PROGRAM ldrMain
VAR


	AIN1 AT %I*: UINT :=0;
	AOUT1 AT %Q*: INT := 1000;
	
	RUNNING: BOOL := FALSE;
	START: BOOL := TRUE;
	
END_VAR
VAR // added by the converter: edge detectors and wires of the graphical bodies
    _w1 : BOOL;
END_VAR

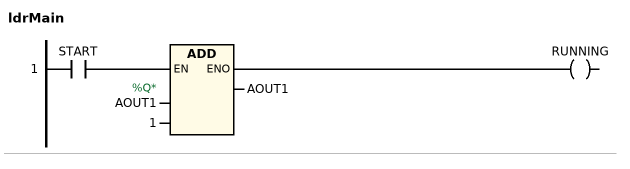
// NETWORK 1
//   AOUT1: AT %Q*
_w1 := START;
IF _w1 THEN AOUT1 := AOUT1 + 1; END_IF
RUNNING := _w1;

END_PROGRAM

(* stored: Version 1.1.0.1, ProductVersion 3.1.0.36
   POU ldrMain: Id {f57934a2-7241-4ecd-ad09-494bcab90e1f}, SpecialFunc None *)
